FUNCTION_BLOCK SpriteSheetAnimationFrames implements I_Animation
VAR
	spriteSheetFilePath : T_MAXSTRING;
	spriteWidth : UDINT;
	spriteHeight : UDINT;
	totalSprites : UDINT;
	columns : UDINT;
	rows : UDINT;
	spriteSheetImage : ITcVnImage;
	readImage: FB_VN_ReadImage;
	
	// animation variables
	_currentFrameIndex : UDINT;
	_currentFrameImage : ITcVnImage;
END_VAR

PROPERTY PUBLIC CurrentFrameImage : ITcVnImage
GET
CurrentFrameImage := _currentFrameImage;
END_GET
END_PROPERTY

PROPERTY PUBLIC CurrentFrameIndex : UDINT
GET
CurrentFrameIndex := _currentFrameIndex;
END_GET
END_PROPERTY

METHOD FB_init : BOOL
VAR_INPUT
	bInitRetains : BOOL; // if TRUE, the retain variables are initialized (warm start / cold start)
	bInCopyCode : BOOL;  // if TRUE, the instance afterwards gets moved into the copy code (online change)
	SpriteSheetFilePath : T_MAXSTRING;
	SpriteWidth : UDINT;
	SpriteHeight : UDINT;
	TotalSprites : UDINT;
	Columns : UDINT;
	Rows : UDINT;
END_VAR
THIS^.spriteSheetFilePath := SpriteSheetFilePath;
THIS^.spriteWidth := SpriteWidth;
THIS^.spriteHeight := SpriteHeight;
THIS^.totalSprites := TotalSprites;
THIS^.columns := Columns;
THIS^.rows := Rows;
END_METHOD

PROPERTY PUBLIC IsAtLastFrame : BOOL
GET
IF TotalFrameCount = 0 THEN
	IsAtLastFrame := TRUE;
	RETURN;
END_IF

IsAtLastFrame := CurrentFrameIndex = TotalFrameCount - 1;
END_GET
END_PROPERTY

METHOD PUBLIC MoveToStart
VAR_INPUT
END_VAR
_currentFrameIndex := 0;
TryGetSprite(_currentFrameIndex, _currentFrameImage);
END_METHOD

PROPERTY PUBLIC TotalFrameCount : UDINT
GET
TotalFrameCount := totalSprites;
END_GET
END_PROPERTY

METHOD PRIVATE TryGetSprite : BOOL
VAR_INPUT
	Index : UDINT;
	Destination : REFERENCE TO ITcVnImage;
END_VAR
VAR
	spriteX : UDINT;
	spriteY : UDINT;
	spriteColumn : UDINT;
	spriteRow : UDINT;
	result : HRESULT;
END_VAR
IF Index > TotalFrameCount - 1 THEN
	RETURN;
END_IF

spriteColumn := Index MOD columns;
spriteRow := Index / columns;

spriteX := spriteColumn * spriteWidth;
spriteY := spriteRow * spriteHeight;

result := F_VN_CopyImage(spriteSheetImage, _currentFrameImage, s_OK);
result := F_VN_SetRoi(spriteX, spriteY, spriteWidth, spriteHeight, _currentFrameImage, result);

TryGetSprite := Succeeded(result);
END_METHOD

METHOD PUBLIC TryLoad : BOOL
VAR
	i : UDINT;
END_VAR
// if we already have an image loaded, then we can early jump out as we know everything is done. 
IF spriteSheetImage <> 0 THEN
	TryLoad := TRUE;
	RETURN;
END_IF

IF spriteSheetFilePath = '' OR  spriteWidth = 0 OR spriteHeight = 0 OR totalSprites = 0 OR columns = 0 OR rows = 0 THEN
	// this is our sanity check, we return out if anything is bad.
	// if we pass this point we know we can use the variables confidently.
	RETURN;
END_IF

// we keep polling the read until an image is read.  If it faults due to error then we just sit here and never return true.
readImage(sFilePath := spriteSheetFilePath, ipDestImage := spriteSheetImage, bRead := TRUE, nTimeout := T#500MS);
IF readImage.bBusy THEN 
	RETURN;
END_IF

IF readImage.bError THEN 
	RETURN;
END_IF 

// at this point we should have an image, so we will do one final check before moving on.  
IF spriteSheetImage = 0 THEN
	RETURN;
END_IF

// we have made it this far, which means we need to set the CurrentFrameImage to the first part of the image and report as done. 
MoveToStart();
TryLoad := TRUE;
END_METHOD

METHOD PUBLIC TryMoveNext : BOOL
VAR_INPUT
END_VAR
IF _currentFrameIndex = TotalFrameCount - 1 THEN
	RETURN;
END_IF

_currentFrameIndex := _currentFrameIndex + 1;
TryMoveNext := TryGetSprite(_currentFrameIndex, _currentFrameImage);
END_METHOD

METHOD PUBLIC TryMovePrevious : BOOL
VAR_INPUT
END_VAR
IF _currentFrameIndex = 0 THEN
	RETURN;
END_IF

_currentFrameIndex := _currentFrameIndex - 1;
TryMovePrevious := TryGetSprite(_currentFrameIndex, _currentFrameImage);
END_METHOD

END_FUNCTION_BLOCK

(* stored: Version 1.1.0.1, ProductVersion 3.1.4024.13
   POU SpriteSheetAnimationFrames: Id {d28c0ddf-ffdd-454b-af0f-acb5bf9aa81a}, SpecialFunc None
   Folder Constructor: Id {2dc1fcc5-fe39-4ab3-990e-a40313008602}
   Folder Private: Id {5f1236e4-977d-4c2b-9f82-917a26ae9917}
   Property CurrentFrameImage: Id {7eed3f1d-24a4-4b7f-807b-e67f3bb2cedf}
   Get Get: Id {d3a9abee-c421-46be-85a4-076d9cb6728a}
   Property CurrentFrameIndex: Id {7ebf164b-8823-4e72-ae20-56d870b0a047}
   Get Get: Id {af68c9a1-eb15-4aa9-a945-317f81d8971d}
   Method FB_init: Id {236f79e8-3370-4e5e-84ba-000dc06437e2}
   Property IsAtLastFrame: Id {a2ed32b5-2a89-414d-bda9-fe3764b0c496}
   Get Get: Id {7c750380-163f-4e9e-b08d-d9ed67a30789}
   Method MoveToStart: Id {f34c7f15-d205-4004-b315-4a1c0e9b3abc}
   Property TotalFrameCount: Id {76fe5976-5bb5-4706-aa9b-a7897641e14a}
   Get Get: Id {28eef738-fec6-4adf-b0c6-83837418330b}
   Method TryGetSprite: Id {daabe6d8-56ff-421e-b74f-0f0902a20d80}
   Method TryLoad: Id {f737a074-84cf-4fbb-8517-d5385a7c987b}
   Method TryMoveNext: Id {6c8107ea-5438-4b15-a392-622897f94951}
   Method TryMovePrevious: Id {f70cba11-7a90-4f06-b745-e52a98c19092} *)
